// TIA Portal V19 export
TYPE "LEXCHANGETRAY_typeHandlingXyzEm_toNgConveyorRecieve"
// stored: Access Published
   STRUCT
      feedback { S7_SetPoint := 'True'} : "LEXCHANGETRAY_typeNgConveyorEm_toHandlingXyzFeedback";
      req { S7_SetPoint := 'True'} : "LEXCHANGETRAY_typeNgConveyorEm_toHandlingXyzReq";
   END_STRUCT;
END_TYPE
